{attribute addProperty BoxType "EJ5002-0000-0016"}
{attribute addProperty Id "StatusAT %I*Status_3D859DDA1621Counter_valueAT %I*UDINT32417"}
{attribute addProperty CRC "4157749457"}
{attribute addProperty SizeInBites "48"}
{attribute addProperty SizeInBytes "6"}
TYPE SSI_Inputs_Channel_F7D238D1 :
STRUCT
	{attribute addProperty Name "Status"}
	Status AT %I* : Status_3D859DDA;
	{attribute addProperty Name "Counter_value"}
	Counter_value AT %I* : UDINT;
END_STRUCT
END_TYPE

(* stored: Version 1.2.0.0, ProductVersion 3.1.4024.9
   DUT SSI_Inputs_Channel_F7D238D1: Id {c57ab24c-a0db-481f-ab5e-1b97eb830c0b} *)
